INTERFACE I_EnumDatatype EXTENDS I_UserDefinedDatatype

END_INTERFACE

(* stored: Version 1.1.0.1, ProductVersion 3.1.4024.12
   Itf I_EnumDatatype: Id {a66f96e8-bffb-017f-0793-23e954ebdfef} *)
